// TIA Portal V20 export
// export: Created 2025-12-01T14:57:12.1026524Z, ExportSetting None, DisplayName Totally Integrated Automation Portal, DisplayVersion V20 Update 3, DisplayName TIA Portal Openness, DisplayVersion V20 Update 3, DisplayName TIA Portal Version Control Interface, DisplayVersion V20 Update 3, DisplayName STEP 7 Professional, DisplayVersion V20 Update 3, DisplayName STEP 7 Safety, DisplayVersion V20 Update 2, DisplayName WinCC Basic/Comfort/Advanced, DisplayVersion V20 Update 3, DisplayName WinCC Professional, DisplayVersion V20 Update 3, DisplayName WinCC Unified, DisplayVersion V20 Update 3
FUNCTION "FC981_CTRL_VAR_MOVIMOT" : Void   // FC981, LAD
{ S7_Optimized_Access := 'FALSE' }
AUTHOR : MOVIMOT
FAMILY : PROFIBUS
NAME : 20130301
VERSION : 3.0
// This sample program shows the basic approach only.
// We do not accept legal or other liability for
// incorrect program functions and their consequences!
// stored: AutoNumber false, SetENOAutomatically false
   VAR_INPUT
      Dir_INI : Int;   // Direccion Inicial de la Palabra de Estado y Control. Misma direccion el en HW.
      Avance : Bool;
      Retroceso : Bool;
      Sentido_Giro : Bool;   // Inversion del sentido de giro.
      RESET : Bool;   // Reseteo del equipo MOVIMOT.
      RELEASE_THE_BRAKE : Bool;   // Desbloquear el freno sin habilitación del accionamiento.
      SETPOINT_SPEED : Int;   // Consigna el valor porcentual: máx. 100%
      RAMP_ms : Int;   // ACC/DCC en milisegundos.
   END_VAR
   VAR_OUTPUT
      INVERTER_READY : Bool;
      FAULT_OF_AXIS : Bool;
      FAULT_NO : Int;
      OUTPUT_CURRENT : Int;   // % de la corriente nominal
   END_VAR
   VAR_TEMP
      PI : Struct
         STATUS : Byte;
         ENABLE_OUTPUT_STAGE : Bool;
         INVERTER_READY : Bool;
         PO_DATA_ENABLE : Bool;
         STW_BIT_3 : Bool;
         STW_BIT_4 : Bool;
         ERROR : Bool;
         STW_BIT_6 : Bool;
         STW_BIT_7 : Bool;
         OUTPUT_CURRENT : Int;
         STW2_BIT_13 : Bool;
         STW2_BIT_14 : Bool;
         STW2_BIT_15 : Bool;
         STW2_BIT_0 : Bool;
         STW2_BIT_1 : Bool;
         STW2_BIT_2 : Bool;
         STW2_BIT_3 : Bool;
         STW2_BIT_4 : Bool;
         ERROR_BIT : Bool;
         STW2_BIT_6 : Bool;
         STW2_BIT_7 : Bool;
      END_STRUCT;
      PO : Struct
         RELEASE_THE_BRAKE : Bool;
         CTW_BIT_9 : Bool;
         CTW_BIT_10 : Bool;
         CTW_BIT_11 : Bool;
         CTW_BIT_12 : Bool;
         CTW_BIT_13 : Bool;
         CTW_BIT_14 : Bool;
         CTW_BIT_15 : Bool;
         CONTR_INHIBIT : Bool;
         RAPID_STOP : Bool;
         STOP : Bool;
         CTW_BIT_3 : Bool;
         CTW_BIT_4 : Bool;
         CTW_BIT_5 : Bool;
         RESET_FAULT : Bool;
         CTW_BIT_7 : Bool;
         SETPOINT_SPEED : Int;
         RAMP : Int;
      END_STRUCT;
      Addr : DWord;
      P_PI : DWord;
      P_PO : DWord;
      PIn_1 : Int;
      PIn_2 : Int;
      PIn_3 : Int;
      Speed_SetPoint : Int;
   END_VAR
   VAR_TEMP   // added for the SCL form of the ladder/FBD networks
      _w1 : Bool;
      _w2 : Bool;
   END_VAR
BEGIN

NETWORK
TITLE = Lectura de datos de la Periferia
// Calculo puntero datos donde vamos a ir recogiendo la información
      L     #Dir_INI;
      SLD   3;  //Dar formato de Integer a Puntero
      LAR1;


//=======================================================================================================================
// Leemos todos los datos de periferia
//Es simualcion??
      A     "Activar_Simulador";
      JC    EnSimulacionLectura;

/// Leer de periferia. No se esta simulando
// Primer Word
      L     IW [AR1, P#0.0];
      T     #PIn_1;

// Segundo Word
      L     IW [AR1, P#2.0];
      T     #PIn_2;

// Tercer Word
      L     IW [AR1, P#4.0];
      T     #PIn_3;
      JU    finLectura;

//En simulacion
EnSimulacionLectura:NOP   0;
// Primer Word
      L     IW [AR1, P#0.0];
      T     #PIn_1;

// Segundo Word
      L     IW [AR1, P#2.0];
      T     #PIn_2;

// Tercer Word
      L     IW [AR1, P#4.0];
      T     #PIn_3;
//////////////////
finLectura:NOP   0;





NETWORK
TITLE = Prepare process input data

      L     P##PI;  // - Puntero
      T     #P_PI;

      L     #PIn_1;
      T     LW [#P_PI];  // LW     0
      L     #PIn_2;
      T     #PI.OUTPUT_CURRENT;

      L     #P_PI;
      L     P#4.0;
      +D;
      T     #P_PI;
      L     #PIn_3;
      T     LW [#P_PI];  // LW     4


      L     #PI.OUTPUT_CURRENT;
      L     10;  //Adapt 1 digit = 0.1% In to 1% In
      /I;
      T     #OUTPUT_CURRENT;

      A     #PI.INVERTER_READY;
      =     #INVERTER_READY;

      A     #PI.ERROR;
      =     #FAULT_OF_AXIS;


REGION Network 3: Evaluate error messages/allocation
   // If an error bit has been set, an error number will be issued.
   // If no error is present, a zero will be issued.
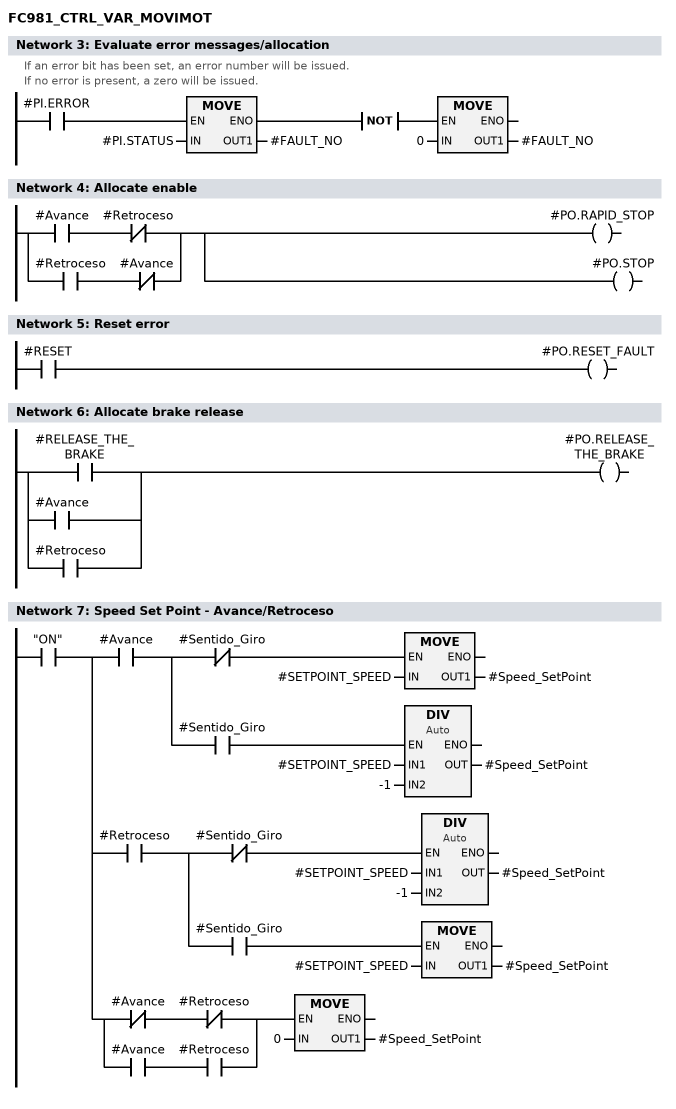
   RUNG wire#powerrail
      Contact( #PI.ERROR )
      { S7_GenerateENO := "TRUE" } Move(in := #PI.STATUS, out1 => #FAULT_NO)
      Not()
      { S7_GenerateENO := "TRUE" } Move(in := 0, out1 => #FAULT_NO)
   END_RUNG
   // the same network as SCL:
   // ENO of a box is taken as its EN; it also drops when the box reports an error
   IF #PI.ERROR THEN #FAULT_NO := #PI.STATUS; END_IF;
   IF NOT #PI.ERROR THEN #FAULT_NO := 0; END_IF;
END_REGION

REGION Network 4: Allocate enable
   RUNG wire#powerrail
      Contact( #Avance )
      I_Contact( #Retroceso )
      wire#w1
      Coil( #PO.RAPID_STOP )
   END_RUNG
   RUNG wire#powerrail
      Contact( #Retroceso )
      I_Contact( #Avance )
   END_RUNG wire#w1
   RUNG wire#w1
      Coil( #PO.STOP )
   END_RUNG
   // the same network as SCL:
   #PO.RAPID_STOP := (#Avance AND NOT #Retroceso) OR (#Retroceso AND NOT #Avance);
   #PO.STOP := #PO.RAPID_STOP;
END_REGION

REGION Network 5: Reset error
   RUNG wire#powerrail
      Contact( #RESET )
      Coil( #PO.RESET_FAULT )
   END_RUNG
   // the same network as SCL:
   #PO.RESET_FAULT := #RESET;
END_REGION

REGION Network 6: Allocate brake release
   RUNG wire#powerrail
      Contact( #RELEASE_THE_BRAKE )
      wire#w1
      Coil( #PO.RELEASE_THE_BRAKE )
   END_RUNG
   RUNG wire#powerrail
      Contact( #Avance )
   END_RUNG wire#w1
   RUNG wire#powerrail
      Contact( #Retroceso )
   END_RUNG wire#w1
   // the same network as SCL:
   #PO.RELEASE_THE_BRAKE := #RELEASE_THE_BRAKE OR #Avance OR #Retroceso;
END_REGION

REGION Network 7: Speed Set Point - Avance/Retroceso
   RUNG wire#powerrail
      Contact( "ON" )
      wire#w1
      Contact( #Avance )
      wire#w2
      I_Contact( #Sentido_Giro )
      { S7_GenerateENO := "TRUE" } Move(in := #SETPOINT_SPEED, out1 => #Speed_SetPoint)
   END_RUNG
   RUNG wire#w2
      Contact( #Sentido_Giro )
      Div(in1 := #SETPOINT_SPEED, in2 := -1, out => #Speed_SetPoint)
   END_RUNG
   RUNG wire#w1
      Contact( #Retroceso )
      wire#w3
      I_Contact( #Sentido_Giro )
      Div(in1 := #SETPOINT_SPEED, in2 := -1, out => #Speed_SetPoint)
   END_RUNG
   RUNG wire#w3
      Contact( #Sentido_Giro )
      { S7_GenerateENO := "TRUE" } Move(in := #SETPOINT_SPEED, out1 => #Speed_SetPoint)
   END_RUNG
   RUNG wire#w1
      I_Contact( #Avance )
      I_Contact( #Retroceso )
      wire#w4
      { S7_GenerateENO := "TRUE" } Move(in := 0, out1 => #Speed_SetPoint)
   END_RUNG
   RUNG wire#w1
      Contact( #Avance )
      Contact( #Retroceso )
   END_RUNG wire#w4
   // the same network as SCL:
   #_w1 := "ON" AND #Avance;
   IF #_w1 AND NOT #Sentido_Giro THEN #Speed_SetPoint := #SETPOINT_SPEED; END_IF;
   IF #_w1 AND #Sentido_Giro THEN #Speed_SetPoint := #SETPOINT_SPEED / (-1); END_IF;
   #_w2 := "ON" AND #Retroceso;
   IF #_w2 AND NOT #Sentido_Giro THEN #Speed_SetPoint := #SETPOINT_SPEED / (-1); END_IF;
   IF #_w2 AND #Sentido_Giro THEN #Speed_SetPoint := #SETPOINT_SPEED; END_IF;
   IF "ON" AND ((NOT #Avance AND NOT #Retroceso) OR (#Avance AND #Retroceso)) THEN
       #Speed_SetPoint := 0;
   END_IF;
END_REGION

NETWORK
TITLE = Prepare process output data
      SET;  //Reset of all control word bits not in use
      R     #PO.CONTR_INHIBIT;
      R     #PO.CTW_BIT_3;
      R     #PO.CTW_BIT_4;
      R     #PO.CTW_BIT_5;
      R     #PO.CTW_BIT_7;

      R     #PO.CTW_BIT_9;
      R     #PO.CTW_BIT_10;
      R     #PO.CTW_BIT_11;
      R     #PO.CTW_BIT_12;
      R     #PO.CTW_BIT_13;
      R     #PO.CTW_BIT_14;
      R     #PO.CTW_BIT_15;


      L     #Speed_SetPoint;  //Adapt set speed: +100% corresponds to 4000hex
      ITD;
      L     DW#16#4000;  //PO.Setpoint_speed = Setpoint_speed * 4000h / 100d
      *D;
      L     DINT#100;
      /D;
      T     #PO.SETPOINT_SPEED;

      L     #RAMP_ms;
      T     #PO.RAMP;

//Calculo puntero datos donde vamos a ir recogiendo la información
      L     #Dir_INI;
      SLD   3;  //Dar formato de Integer a Puntero
      LAR1;
//Es simualcion??
      A     "Activar_Simulador";
      JC    EnSimulacion;
//pasar los valores de los temporales a la periferia y a las salidas de la funcion.
// temp.PO -> Periferia de salida
      L     P##PO;  // - Puntero
      T     #P_PO;

      L     LW [#P_PO];  //cargamos el PO
      T     QW [AR1, P#0.0];  // Primer Word

      L     #PO.SETPOINT_SPEED;
      T     QW [AR1, P#2.0];  // Segundo Word

      L     #PO.RAMP;
      T     QW [AR1, P#4.0];  // Tercer Word
      JU    fin;
EnSimulacion:NOP   0;
//pasar los valores de los temporales a la periferia y a las salidas de la funcion.
// temp.PO -> Periferia de salida
      L     P##PO;  // - Puntero
      T     #P_PO;

      L     LW [#P_PO];  //cargamos el PO
      T     QW [AR1, P#0.0];  // Primer Word

      L     #PO.SETPOINT_SPEED;
      T     QW [AR1, P#2.0];  // Segundo Word

      L     #PO.RAMP;
      T     QW [AR1, P#4.0];  // Tercer Word
fin:  NOP   0;
END_FUNCTION
